SYSTEM X2Y2_TESTR (* System Configuration to test X2Y2 with RMT_FRAME *)
  (* Standard: 61499-1 *)
  (* Version 0.0, 2003-08-13, JHC, Rockwell Automation, Adapted from X2Y2_TESTD *)
  APPLICATION APP1 (* Testing FB_X2Y2 *)
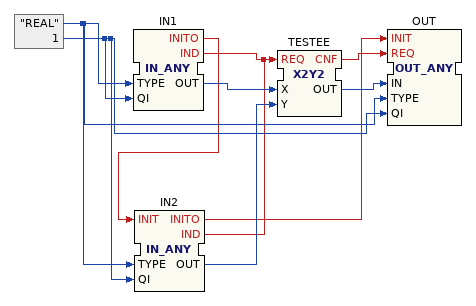
    FBS
      IN1 : IN_ANY;
      IN2 : IN_ANY;
      TESTEE : X2Y2;
      OUT : OUT_ANY;
    END_FBS
    EVENT_CONNECTIONS
      IN1.INITO TO IN2.INIT;
      IN2.INITO TO OUT.INIT;
      IN1.IND TO TESTEE.REQ;
      IN2.IND TO TESTEE.REQ;
      TESTEE.CNF TO OUT.REQ;
    END_CONNECTIONS
    DATA_CONNECTIONS
      IN1.OUT TO TESTEE.X;
      IN2.OUT TO TESTEE.Y;
      TESTEE.OUT TO OUT.IN;
      "REAL" TO IN2.TYPE;
      "REAL" TO OUT.TYPE;
      "REAL" TO IN1.TYPE;
      1 TO IN1.QI;
      1 TO IN2.QI;
      1 TO OUT.QI;
    END_CONNECTIONS
  END_APPLICATION
  DEVICE DEV1 : FRAME_DEVICE
    RESOURCE RES1 : PANEL_RESOURCE
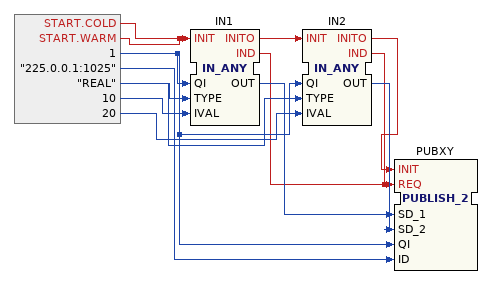
      FBS
        IN1 : IN_ANY;
        IN2 : IN_ANY;
        PUBXY : PUBLISH_2;
      END_FBS
      EVENT_CONNECTIONS
        START.COLD TO IN1.INIT;
        START.WARM TO IN1.INIT;
        IN1.INITO TO IN2.INIT;
        IN2.INITO TO PUBXY.INIT;
        IN1.IND TO PUBXY.REQ;
        IN2.IND TO PUBXY.REQ;
      END_CONNECTIONS
      DATA_CONNECTIONS
        1 TO IN1.QI;
        1 TO IN2.QI;
        IN1.OUT TO PUBXY.SD_1;
        IN2.OUT TO PUBXY.SD_2;
        1 TO PUBXY.QI;
        "225.0.0.1:1025" TO PUBXY.ID;
        "REAL" TO IN1.TYPE;
        10 TO IN1.IVAL;
        "REAL" TO IN2.TYPE;
        20 TO IN2.IVAL;
      END_CONNECTIONS
    END_RESOURCE
  END_DEVICE
  DEVICE DEV2 : RMT_FRAME
    RESOURCE RES2 : PANEL_RESOURCE
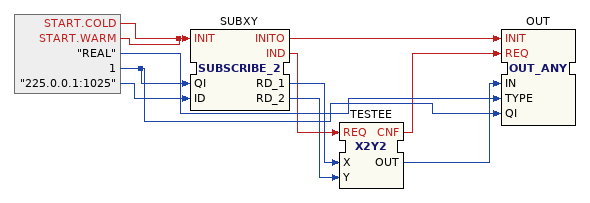
      FBS
        SUBXY : SUBSCRIBE_2;
        TESTEE : X2Y2;
        OUT : OUT_ANY;
      END_FBS
      EVENT_CONNECTIONS
        START.COLD TO SUBXY.INIT;
        START.WARM TO SUBXY.INIT;
        SUBXY.INITO TO OUT.INIT;
        SUBXY.IND TO TESTEE.REQ;
        TESTEE.CNF TO OUT.REQ;
      END_CONNECTIONS
      DATA_CONNECTIONS
        TESTEE.OUT TO OUT.IN;
        "REAL" TO OUT.TYPE;
        1 TO OUT.QI;
        1 TO SUBXY.QI;
        SUBXY.RD_1 TO TESTEE.X;
        SUBXY.RD_2 TO TESTEE.Y;
        "225.0.0.1:1025" TO SUBXY.ID;
      END_CONNECTIONS
    END_RESOURCE
  END_DEVICE
  DATA_CONNECTIONS (* parameter values *)
    [150,150,125,100] TO DEV1.BOUNDS;
    [1,1] TO DEV1.GRID;
    [150,250,125,75] TO DEV2.BOUNDS;
    [1,1] TO DEV2.GRID;
  END_CONNECTIONS
  MAPPINGS
    APP1.IN1 ON DEV1.RES1.IN1;
    APP1.IN2 ON DEV1.RES1.IN2;
    APP1.TESTEE ON DEV2.RES2.TESTEE;
    APP1.OUT ON DEV2.RES2.OUT;
  END_MAPPINGS
END_SYSTEM
